SUBAPPLICATION Uebung_104_AX (* Zustandsbasierte Schrittkette mit Power-Fail Recovery (AX-Version) *)
  (* Standard: 61499-2; Description: Copyright (c) 2026 HR Agrartechnik GmbH This program and the accompanying materials are made available under the terms of the Eclipse Public License 2.0 which is available at https://www.eclipse.org/legal/epl-2.0/ SPDX-License-Identifier: EPL-2.0 *)
  (* Version 1.0, 2026-04-20, Franz Höpfinger, HR Agrartechnik GmbH, initial API and implementation *)
  PACKAGE Uebungen;
  IMPORT logiBUS::io::DI::logiBUS_DI::Input_I1;
  IMPORT logiBUS::io::DI::logiBUS_DI::Input_I2;
  IMPORT logiBUS::io::DI::logiBUS_DI::Input_I3;
  IMPORT logiBUS::io::DI::logiBUS_DI::Input_I4;
  IMPORT logiBUS::io::DQ::logiBUS_DO::Output_Q1;
  IMPORT logiBUS::io::DQ::logiBUS_DO::Output_Q2;
  IMPORT logiBUS::io::DQ::logiBUS_DO::Output_Q3;
  IMPORT logiBUS::io::DQ::logiBUS_DO::Output_Q4;
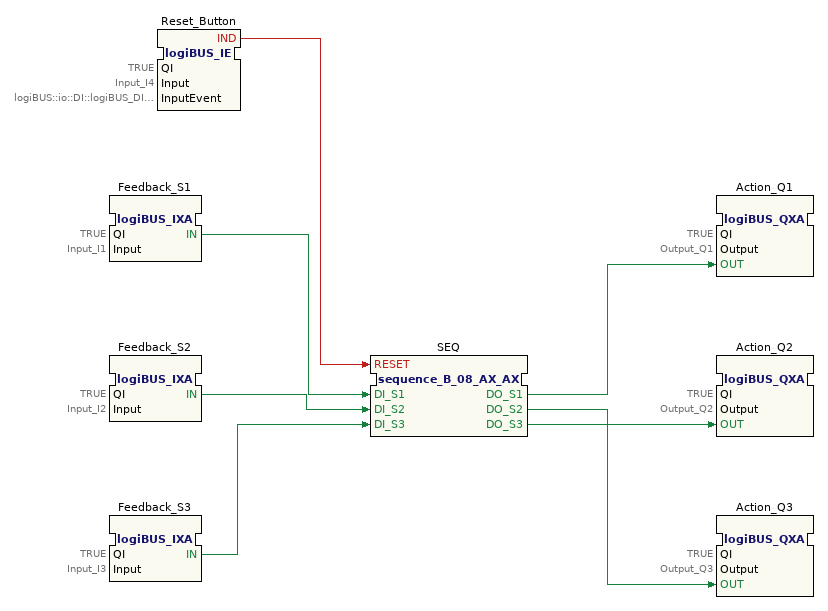
  (* Diese Schrittkette springt beim Einschalten direkt in den Zustand, dessen Eingangs-Adapter auf TRUE steht (Recovery). *)
  FBS
    SEQ : logiBUS::utils::sequence::boolean::sequence_B_08_AX_AX;
    Feedback_S1 : logiBUS::io::DI::logiBUS_IXA(QI := TRUE, Input := Input_I1);
    Feedback_S2 : logiBUS::io::DI::logiBUS_IXA(QI := TRUE, Input := Input_I2);
    Feedback_S3 : logiBUS::io::DI::logiBUS_IXA(QI := TRUE, Input := Input_I3);
    Reset_Button : logiBUS::io::DI::logiBUS_IE(QI := TRUE, Input := Input_I4, InputEvent := logiBUS::io::DI::logiBUS_DI_Events::BUTTON_SINGLE_CLICK);
    Action_Q1 : logiBUS::io::DQ::logiBUS_QXA(QI := TRUE, Output := Output_Q1);
    Action_Q2 : logiBUS::io::DQ::logiBUS_QXA(QI := TRUE, Output := Output_Q2);
    Action_Q3 : logiBUS::io::DQ::logiBUS_QXA(QI := TRUE, Output := Output_Q3);
  END_FBS
  EVENT_CONNECTIONS
    Reset_Button.IND TO SEQ.RESET;
  END_CONNECTIONS
  ADAPTER_CONNECTIONS
    Feedback_S1.IN TO SEQ.DI_S1;
    Feedback_S2.IN TO SEQ.DI_S2;
    Feedback_S3.IN TO SEQ.DI_S3;
    SEQ.DO_S1 TO Action_Q1.OUT;
    SEQ.DO_S2 TO Action_Q2.OUT;
    SEQ.DO_S3 TO Action_Q3.OUT;
  END_CONNECTIONS
END_SUBAPPLICATION
